# EPICS substitutions: vme_iocs/iocbio4/iocBoot/motor.substitutions
file "$(MOTOR)/db/motor.db"
{
pattern
{P,		N,	M,		DTYP,			C,	S,	DESC,			EGU,		DIR,	VELO,	VBAS,	ACCL,	BDST,	BVEL,	BACC,	MRES,	PREC,	DHLM,	DLLM,	INIT}
{18ID:,	1,	"m$(N)",	"OMS VME8/44",	0,	0,	"M0X",			mm,			Pos,	1,		.1,		.2,		0,		1,		.2,		2.5e-4,	5,		100,	-100,	""}
{18ID:,	2,	"m$(N)",	"OMS VME8/44",	0,	1,	"M0Y",			mm,			Pos,	1,		.1,		.2,		0,		1,		.2,		2.5e-4,	5,		100,	-100,	""}
{18ID:,	3,	"m$(N)",	"OMS VME8/44",	0,	2,	"M1Y",			mm,			Pos,	1,		.1,		.2,		0,		1,		.2,		2.5e-4,	5,		100,	-100,	""}
{18ID:,	4,	"m$(N)",	"OMS VME8/44",	0,	3,	"M2X",			mm,			Pos,	1,		.1,		.2,		0,		1,		.2,		2.5e-4,	5,		100,	-100,	""}
{18ID:,	5,	"m$(N)",	"OMS VME8/44",	0,	4,	"M2Y",			mm,			Pos,	1,		.1,		.2,		0,		1,		.2,		2.5e-4,	5,		100,	-100,	""}
{18ID:,	6,	"m$(N)",	"OMS VME8/44",	0,	5,	"M2Z",			mm,			Pos,	1,		.1,		.2,		0,		1,		.2,		2.5e-4,	5,		100,	-100,	""}
{18ID:,	7,	"m$(N)",	"OMS VME8/44",	0,	6,	"motor $(N)",	degrees,	Pos,	1,		.1,		.2,		0,		1,		.2,		2.5e-4,	5,		100,	-100,	""}
{18ID:,	8,	"m$(N)",	"OMS VME8/44",	0,	7,	"motor $(N)",	degrees,	Pos,	1,		.1,		.2,		0,		1,		.2,		2.5e-4,	5,		100,	-100,	""}
{18ID:,	9,	"m$(N)",	"OMS VME58",	0,	0,	"motor $(N)",	degrees,	Pos,	1,		.1,		.2,		0,		1,		.2,		2.5e-4,	5,		100,	-100,	""}
{18ID:,	10,	"m$(N)",	"OMS VME58",	0,	1,	"motor $(N)",	degrees,	Pos,	1,		.1,		.2,		0,		1,		.2,		2.5e-4,	5,		100,	-100,	""}
{18ID:,	11,	"m$(N)",	"OMS VME58",	0,	2,	"motor $(N)",	degrees,	Pos,	1,		.1,		.2,		0,		1,		.2,		2.5e-4,	5,		100,	-100,	""}
{18ID:,	12,	"m$(N)",	"OMS VME58",	0,	3,	"motor $(N)",	degrees,	Pos,	1,		.1,		.2,		0,		1,		.2,		2.5e-4,	5,		100,	-100,	""}
{18ID:,	13,	"m$(N)",	"OMS VME58",	0,	4,	"motor $(N)",	degrees,	Pos,	1,		.1,		.2,		0,		1,		.2,		2.5e-4,	5,		100,	-100,	""}
{18ID:,	14,	"m$(N)",	"OMS VME58",	0,	5,	"motor $(N)",	degrees,	Pos,	1,		.1,		.2,		0,		1,		.2,		2.5e-4,	5,		100,	-100,	""}
{18ID:,	15,	"m$(N)",	"OMS VME58",	0,	6,	"motor $(N)",	degrees,	Pos,	1,		.1,		.2,		0,		1,		.2,		2.5e-4,	5,		100,	-100,	""}
{18ID:,	16,	"m$(N)",	"OMS VME58",	0,	7,	"motor $(N)",	degrees,	Pos,	1,		.1,		.2,		0,		1,		.2,		2.5e-4,	5,		100,	-100,	""}
}
